// TIA Portal V17 export
// export: Created 2024-09-02T12:49:54.9851264Z, ExportSetting WithDefaults, DisplayName Totally Integrated Automation Portal, DisplayVersion V17, DisplayName TIA Portal Openness, DisplayVersion V17, DisplayName TIA Portal Version Control Interface, DisplayVersion V17, DisplayName STEP 7 Professional, DisplayVersion V17, DisplayName STEP 7 Safety, DisplayVersion V17, DisplayName WinCC Professional, DisplayVersion V17
FUNCTION "SysFC_FunctionAnalyze" : Void   // FC255, LAD
TITLE = Counter functions / Zaehler Funktionen
{ S7_Optimized_Access := 'TRUE' }
AUTHOR : OlegFuehrus
FAMILY : HMI
NAME : HMI
VERSION : 1.0
// stored: AutoNumber false, IsIECCheckEnabled false, SetENOAutomatically false, UDAEnableTagReadback false
   VAR_INPUT
      i_Start : Bool;   // Auswertung starten / Start evaluation
   END_VAR
   VAR_OUTPUT
      o_Function_active : Bool;   // mindestens eine Funktion aktiv / At least one function active
      o_Num_of_Functions_active : Int;   // Anzahl der aktiven Funktionen / Number of active functions
   END_VAR
   VAR_IN_OUT
      io_Functions : "TypeFunction";
   END_VAR
   VAR_TEMP
      t_Pointer : Int;
   END_VAR
BEGIN

REGION Network 1: INIT
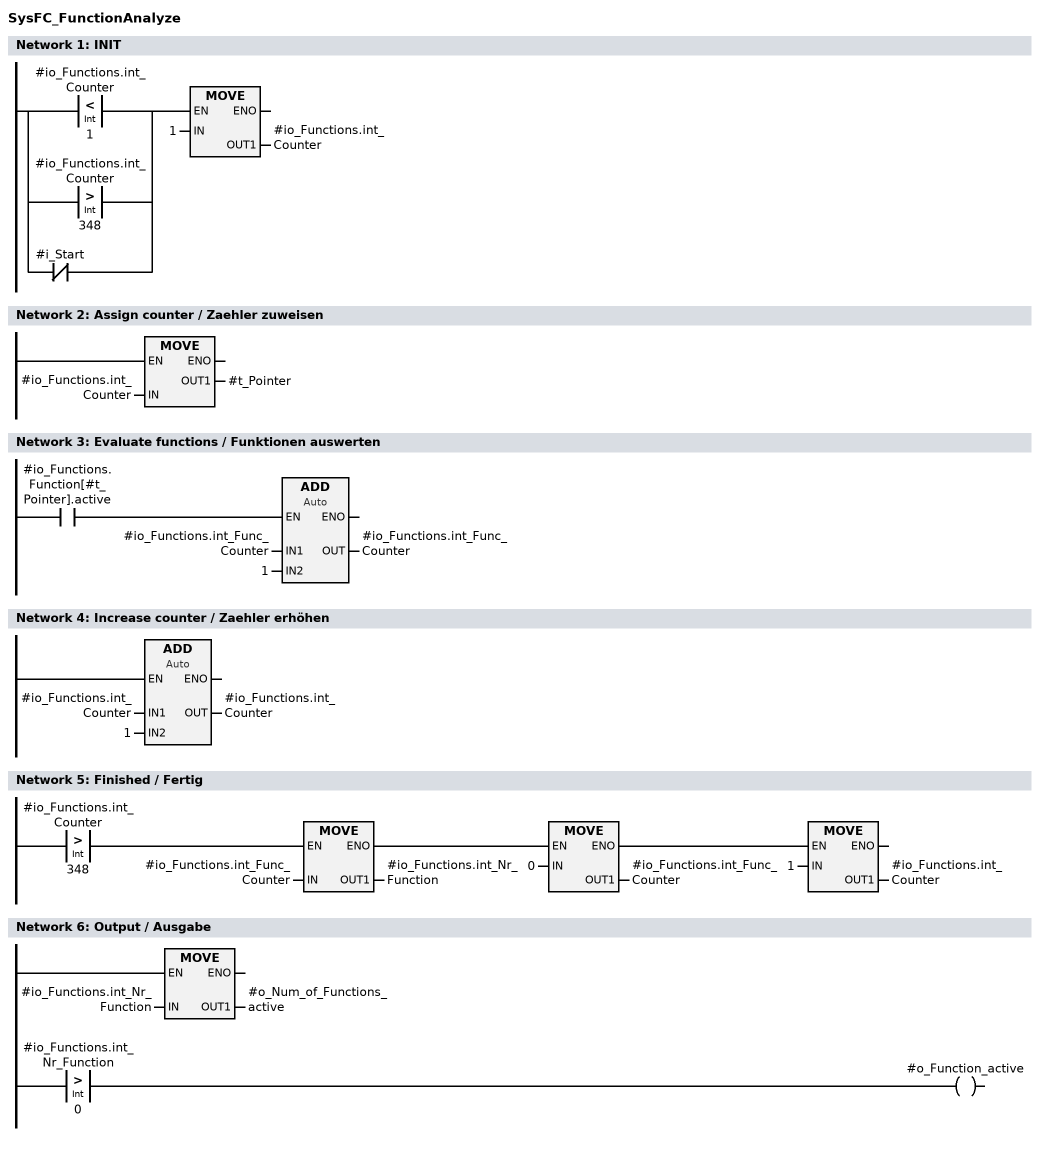
   RUNG wire#powerrail
      { S7_Templates := "SrcType := Int" } LT_Contact(in1 := #io_Functions.int_Counter, in2 := 1)
      wire#w1
      Move(in := 1, out1 => #io_Functions.int_Counter)
   END_RUNG
   RUNG wire#powerrail
      { S7_Templates := "SrcType := Int" } GT_Contact(in1 := #io_Functions.int_Counter, in2 := 348)
   END_RUNG wire#w1
   RUNG wire#powerrail
      I_Contact( #i_Start )
   END_RUNG wire#w1
   // the same network as SCL:
   IF (#io_Functions.int_Counter < 1) OR (#io_Functions.int_Counter > 348) OR NOT #i_Start THEN
       #io_Functions.int_Counter := 1;
   END_IF;
END_REGION

REGION Network 2: Assign counter / Zaehler zuweisen
   RUNG wire#powerrail
      Move(in := #io_Functions.int_Counter, out1 => #t_Pointer)
   END_RUNG
   // the same network as SCL:
   #t_Pointer := #io_Functions.int_Counter;
END_REGION

REGION Network 3: Evaluate functions / Funktionen auswerten
   RUNG wire#powerrail
      Contact( #io_Functions.Function[#t_Pointer].active )
      Add(in1 := #io_Functions.int_Func_Counter, in2 := 1, out => #io_Functions.int_Func_Counter)
   END_RUNG
   // the same network as SCL:
   IF #io_Functions.Function[#t_Pointer].active THEN
       #io_Functions.int_Func_Counter := #io_Functions.int_Func_Counter + 1;
   END_IF;
END_REGION

REGION Network 4: Increase counter / Zaehler erhöhen
   RUNG wire#powerrail
      Add(in1 := #io_Functions.int_Counter, in2 := 1, out => #io_Functions.int_Counter)
   END_RUNG
   // the same network as SCL:
   #io_Functions.int_Counter := #io_Functions.int_Counter + 1;
END_REGION

REGION Network 5: Finished / Fertig
   RUNG wire#powerrail
      { S7_Templates := "SrcType := Int" } GT_Contact(in1 := #io_Functions.int_Counter, in2 := 348)
      Move(in := #io_Functions.int_Func_Counter, out1 => #io_Functions.int_Nr_Function)
      Move(in := 0, out1 => #io_Functions.int_Func_Counter)
      Move(in := 1, out1 => #io_Functions.int_Counter)
   END_RUNG
   // the same network as SCL:
   IF #io_Functions.int_Counter > 348 THEN
       #io_Functions.int_Nr_Function := #io_Functions.int_Func_Counter;
       #io_Functions.int_Func_Counter := 0;
       #io_Functions.int_Counter := 1;
   END_IF;
END_REGION

REGION Network 6: Output / Ausgabe
   RUNG wire#powerrail
      Move(in := #io_Functions.int_Nr_Function, out1 => #o_Num_of_Functions_active)
   END_RUNG
   RUNG wire#powerrail
      { S7_Templates := "SrcType := Int" } GT_Contact(in1 := #io_Functions.int_Nr_Function, in2 := 0)
      Coil( #o_Function_active )
   END_RUNG
   // the same network as SCL:
   #o_Num_of_Functions_active := #io_Functions.int_Nr_Function;
   #o_Function_active := #io_Functions.int_Nr_Function > 0;
END_REGION

REGION Network 7: END / ENDE
END_REGION
END_FUNCTION
